INTERFACE I_SessionManager

METHOD PUBLIC CreateSession : T_MAXSTRING
END_METHOD

METHOD PUBLIC DisposeAllSessions
VAR_INPUT
END_VAR
END_METHOD

METHOD PUBLIC IsValidSession : BOOL
VAR_INPUT
	Id : T_MAXSTRING;
END_VAR
END_METHOD

METHOD PUBLIC RefreshSession
VAR_INPUT
	Id : T_MAXSTRING;
END_VAR
END_METHOD

END_INTERFACE

(* stored: Version 1.1.0.1, ProductVersion 3.1.4024.12
   Itf I_SessionManager: Id {4165cfd1-a2ae-417f-affc-56dd24540fd3}
   Method CreateSession: Id {fed8429b-f1e9-425f-9d52-c3bfdab16c2e}
   Method DisposeAllSessions: Id {e99c1bc0-52ee-4ebf-9f0d-c300e9daf045}
   Method IsValidSession: Id {69f48a35-99ca-4305-9239-5bbb4b6b7d0b}
   Method RefreshSession: Id {9703b05e-fc33-4ea6-a9e0-e38e51a6a160} *)
